Staubli VAL3: naKroznik.pgx

program naKroznik()
begin

  // TUKAJ vstavi ukaze za premikanje robota na krožnik
  // lahko si pomagaš s starimi točkami, ki so tu spodaj zakomentirane

  // namesto mNomSpeed uporabi že pripravljene hitrosti mPočasi, mSrednje in mHitro, glede na to kakšno gibanje želiš
  // ukaz waitEndMove uporabimo, ko želimo, da se robot v vsaki točki ustavi. Ko se pomikamo po prostoru, ne želimo ustavljanja preko vseh točk, ampak želimo zvezno gibanje
  // v definiciji vsake hitrosti je tudi možnost blend, ki pove koliko milimetrov od točke naj potuje robot, ko gre proti naslednji brez ustavljanja
  // če želimo točne pomike, za primer pobiranja, uporabimo waitEndMove, da se robot pomakne točno v točko in tam počaka na naslednji ukaz

  // če podatek ni shranjen kot array (ima le indeks [0]), ga lahko kličemo le z imenom, brez indeksa. Če imamo array z več vnosi/indeksi pa na ta način kličemo ničti [0] element.
  // primer: mNomSpeed[0] == mNomSpeed

  nTaskWorking = nTaskWorking + 1

  movej(jNadPosodo,flange,mSrednje)
  waitEndMove()

  movel(pPoberiPal[0],tLopatka,mSrednje)
  movel(pPoberiPal[1],tLopatka,mSrednje)
  movel(pPoberiPal[2],tLopatka,mPocasi)
  movel(pPoberiPal[3],tLopatka,mPocasi)

  movel(pNaKroznik[0],tLopatka,mPocasi)
  movel(pNaKroznik[1],tLopatka,mPocasi)
  movel(pNaKroznik[2],tLopatka,mSrednje)
  waitEndMove()
  call cakajProgress(3)

  movej(jHome,flange,mSrednje)
  movel(pZajem[2],tSefla,mSrednje)
  waitEndMove()

 nTaskWorking = nTaskWorking - 1
end
